# EPICS SNL sequencer program: viocs/ts_ps/ts_psApp/src/ps_sp_init.stt
program ps_sp_init

int event_proc;
assign event_proc to "EVENT-TSPS-SP-INIT.PROC";

ss ss1 {
    state init {
        when (delay(3.0)) {
            event_proc = 1;
            pvPut(event_proc);
        } exit
    }
}
